% RSLogix 500 project Backwash Alarm Control and Interlock System.RSS, saved by version 9.00.00.04 %
PROJECT "SAMPLE2"    % processor: MicroLogix 1400 %

PROGRAM FILES
  LAD 2 "MAIN"  21 rungs
  LAD 3 "REGEN"  29 rungs
  LAD 4 "FLOW AB"  43 rungs
  LAD 5 "ALARMS"  22 rungs
  LAD 6 "TIME TRIG"  17 rungs  % TIME INTERVAL REGN INITIATION %
  LAD 7 "A VESSEL"  38 rungs
  LAD 8 "ANALOG IN"  6 rungs
  LAD 9 "PRESSURE"  11 rungs
  LAD 10 "B VESSEL"  38 rungs
  LAD 11 "DIGITAL IN"  4 rungs
  LAD 12 "WELL PUMP"  4 rungs
  LAD 16 "DIGITL OUT"  15 rungs
  LAD 17 "REGEN A"  17 rungs
  LAD 18 "REGEN B"  17 rungs
  LAD 19 "RECYCLE"  17 rungs

DATA FILES
  O0 OUTPUT  7 elements
  I1 INPUT  22 elements
  S2 STATUS  66 elements
  B3 COMMON  14 elements
  T4 TIMER  56 elements
  C5 COUNTER  13 elements
  R6 CONTROL  1 elements
  N7   52 elements
  F8 FLOAT  122 elements
  B9 GENCTRL  3 elements
  C10   5 elements
  B21 A  BITS  7 elements
  B22 B BITS  7 elements
  N34   92 elements

LADDER 2 "MAIN"
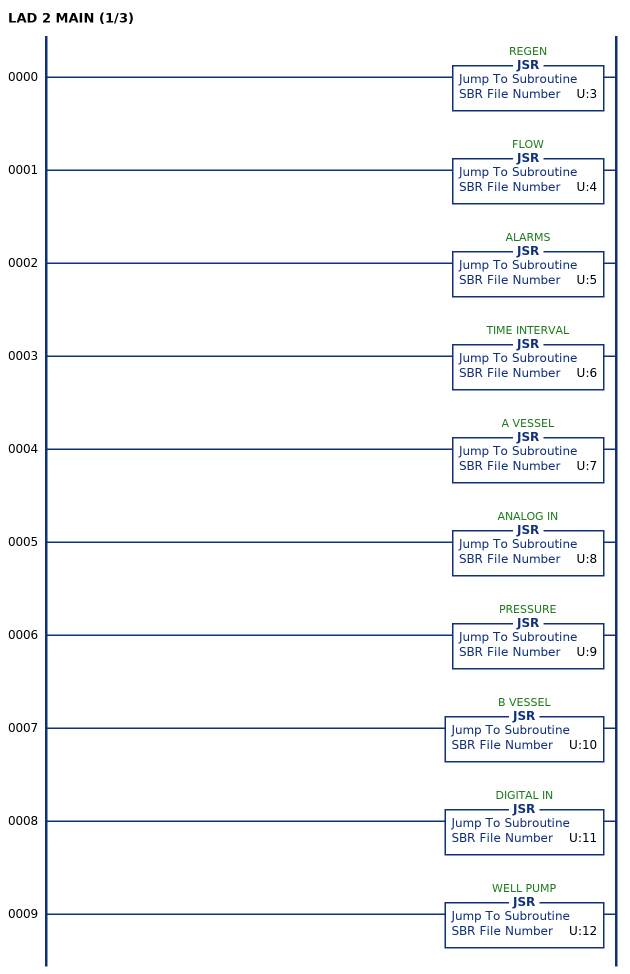
% Rung: 0 %
SOR JSR U:3 EOR
%   U:3  "REGEN" %
% Rung: 1 %
SOR JSR U:4 EOR
%   U:4  "FLOW" %
% Rung: 2 %
SOR JSR U:5 EOR
%   U:5  "ALARMS" %
% Rung: 3 %
SOR JSR U:6 EOR
%   U:6  "TIME INTERVAL" %
% Rung: 4 %
SOR JSR U:7 EOR
%   U:7  "A VESSEL" %
% Rung: 5 %
SOR JSR U:8 EOR
%   U:8  "ANALOG IN" %
% Rung: 6 %
SOR JSR U:9 EOR
%   U:9  "PRESSURE" %
% Rung: 7 %
SOR JSR U:10 EOR
%   U:10  "B VESSEL" %
% Rung: 8 %
SOR JSR U:11 EOR
%   U:11  "DIGITAL IN" %
% Rung: 9 %
SOR JSR U:12 EOR
%   U:12  "WELL PUMP" %

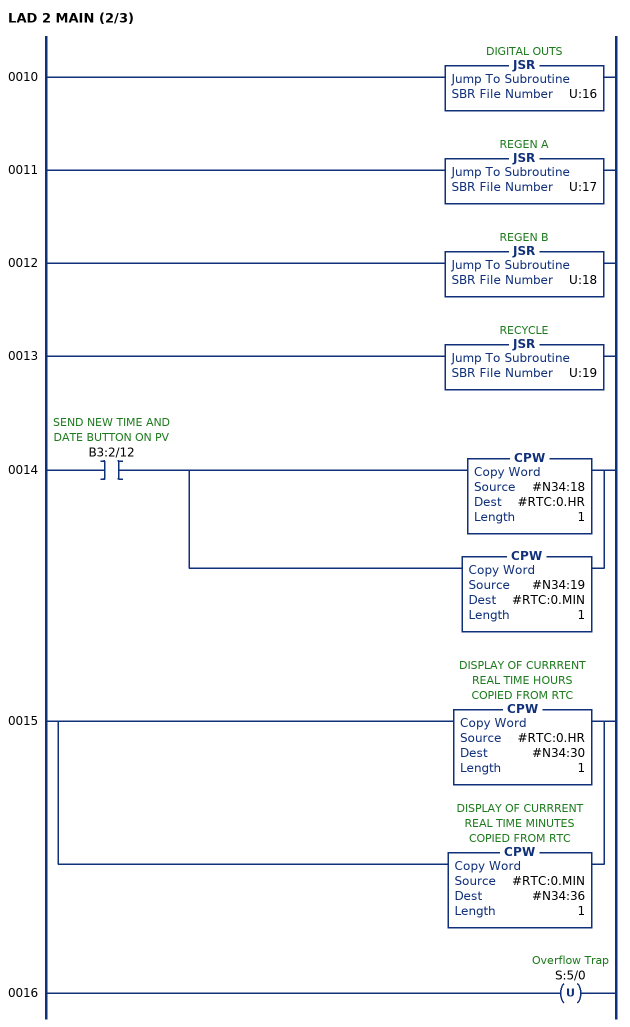
% Rung: 10 %
SOR JSR U:16 EOR
%   U:16  "DIGITAL OUTS" %
% Rung: 11 %
SOR JSR U:17 EOR
%   U:17  "REGEN A" %
% Rung: 12 %
SOR JSR U:18 EOR
%   U:18  "REGEN B" %
% Rung: 13 %
SOR JSR U:19 EOR
%   U:19  "RECYCLE" %
% Rung: 14 %
SOR XIC B3:2/12 BST CPW #N34:18 #RTC:0.HR 1 NXB CPW #N34:19 #RTC:0.MIN 1 BND EOR
%   B3:2/12  "SEND NEW TIME AND DATE BUTTON ON PV" %
%   N34:18  "HOUR INPUT FROM PV" %
%   N34:19  "MINUTE INPUT FROM PV" %
% Rung: 15 %
SOR BST CPW #RTC:0.HR #N34:30 1 NXB CPW #RTC:0.MIN #N34:36 1 BND EOR
%   N34:30  "DISPLAY OF CURRRENT REAL TIME HOURS COPIED FROM RTC" %
%   N34:36  "DISPLAY OF CURRRENT REAL TIME MINUTES COPIED FROM RTC" %
% Rung: 16 %
SOR OTU S:5/0 EOR
%   S:5/0  "Overflow Trap" %

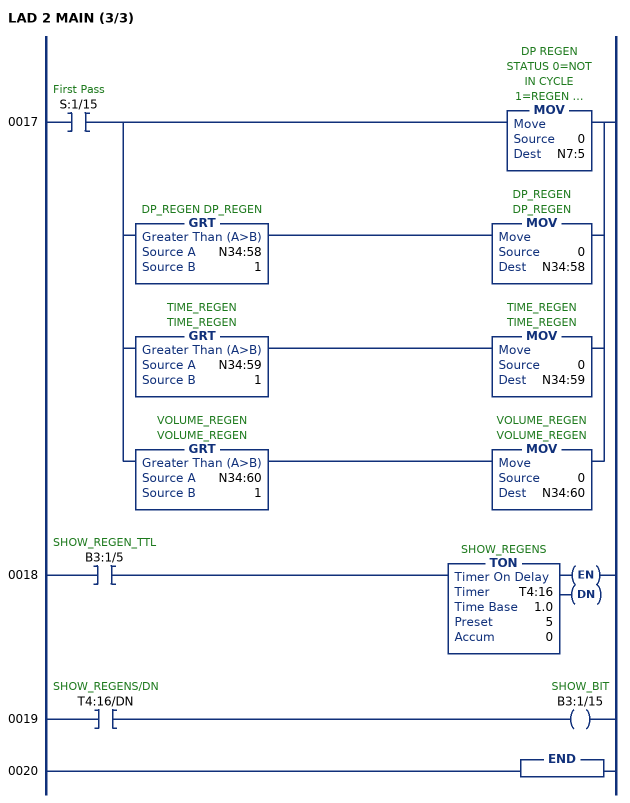
% Rung: 17 %
SOR XIC S:1/15 BST MOV 0 N7:5 NXB GRT N34:58 1 MOV 0 N34:58 NXB GRT N34:59 1 MOV 0 N34:59 NXB GRT N34:60 1 MOV 0 N34:60 BND EOR
%   S:1/15  "First Pass" %
%   N7:5  "DP REGEN STATUS 0=NOT IN CYCLE 1=REGEN A 2=REGEN B" %
%   N34:58  DP_REGEN  "DP_REGEN" %
%   N34:59  TIME_REGEN  "TIME_REGEN" %
%   N34:60  VOLUME_REGEN  "VOLUME_REGEN" %
% Rung: 18 %
SOR XIC B3:1/5 TON T4:16 1.0 5 0 EOR
%   B3:1/5  SHOW_REGEN_TTL %
%   T4:16  SHOW_REGENS %
% Rung: 19 %
SOR XIC T4:16/DN OTE B3:1/15 EOR
%   T4:16  SHOW_REGENS %
%   B3:1/15  SHOW_BIT %
% Rung: 20 %
SOR END EOR

LADDER 3 "REGEN"
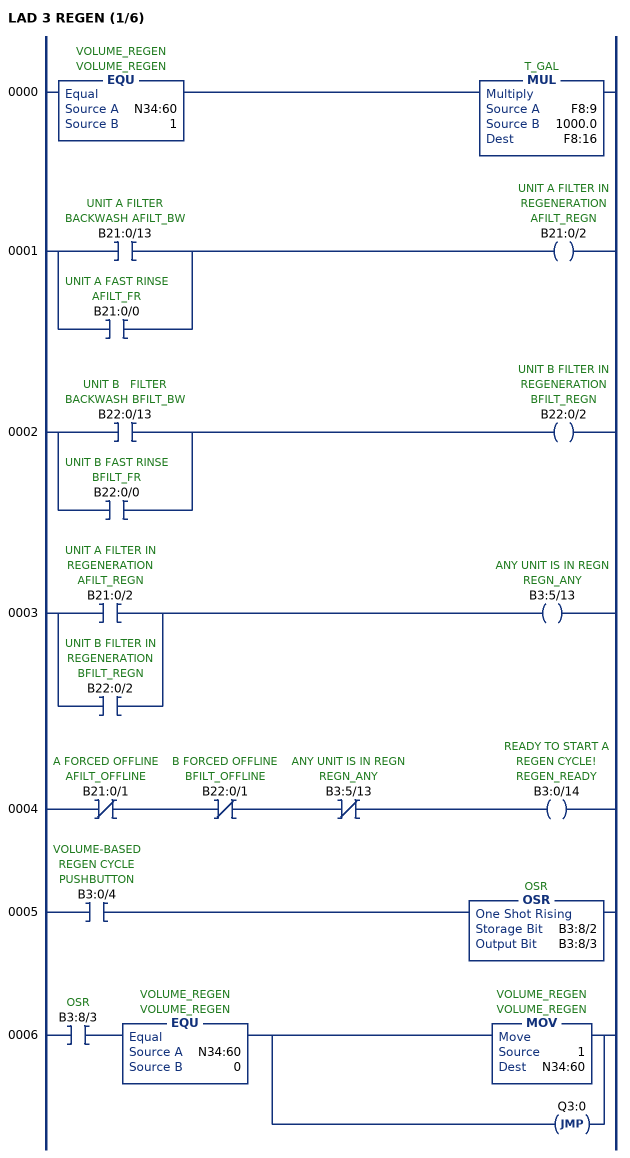
% Rung: 0 %
SOR EQU N34:60 1 MUL F8:9 1000.0 F8:16 EOR
%   N34:60  VOLUME_REGEN  "VOLUME_REGEN" %
%   F8:9  "BATCH ENTRY FOR BATCH START" %
%   F8:16  T_GAL %
% Rung: 1 %
SOR BST XIC B21:0/13 NXB XIC B21:0/0 BND OTE B21:0/2 EOR
%   B21:0/13  AFILT_BW  "UNIT A FILTER BACKWASH" %
%   B21:0/0  AFILT_FR  "UNIT A FAST RINSE" %
%   B21:0/2  AFILT_REGN  "UNIT A FILTER IN REGENERATION" %
% Rung: 2 %
SOR BST XIC B22:0/13 NXB XIC B22:0/0 BND OTE B22:0/2 EOR
%   B22:0/13  BFILT_BW  "UNIT B   FILTER BACKWASH" %
%   B22:0/0  BFILT_FR  "UNIT B FAST RINSE" %
%   B22:0/2  BFILT_REGN  "UNIT B FILTER IN REGENERATION" %
% Rung: 3 %
SOR BST XIC B21:0/2 NXB XIC B22:0/2 BND OTE B3:5/13 EOR
%   B21:0/2  AFILT_REGN  "UNIT A FILTER IN REGENERATION" %
%   B22:0/2  BFILT_REGN  "UNIT B FILTER IN REGENERATION" %
%   B3:5/13  REGN_ANY  "ANY UNIT IS IN REGN" %
% Rung: 4 %
SOR XIO B21:0/1 XIO B22:0/1 XIO B3:5/13 OTE B3:0/14 EOR
%   B21:0/1  AFILT_OFFLINE  "A FORCED OFFLINE" %
%   B22:0/1  BFILT_OFFLINE  "B FORCED OFFLINE" %
%   B3:5/13  REGN_ANY  "ANY UNIT IS IN REGN" %
%   B3:0/14  REGEN_READY  "READY TO START A REGEN CYCLE!" %
% Rung: 5 %
SOR XIC B3:0/4 OSR B3:8/2 B3:8/3 EOR
%   B3:0/4  "VOLUME-BASED REGEN CYCLE PUSHBUTTON" %
%   B3:8/2  "OSR" %
%   B3:8/3  "OSR" %
% Rung: 6 %
SOR XIC B3:8/3 EQU N34:60 0 BST MOV 1 N34:60 NXB JMP Q3:0 BND EOR
%   B3:8/3  "OSR" %
%   N34:60  VOLUME_REGEN  "VOLUME_REGEN" %

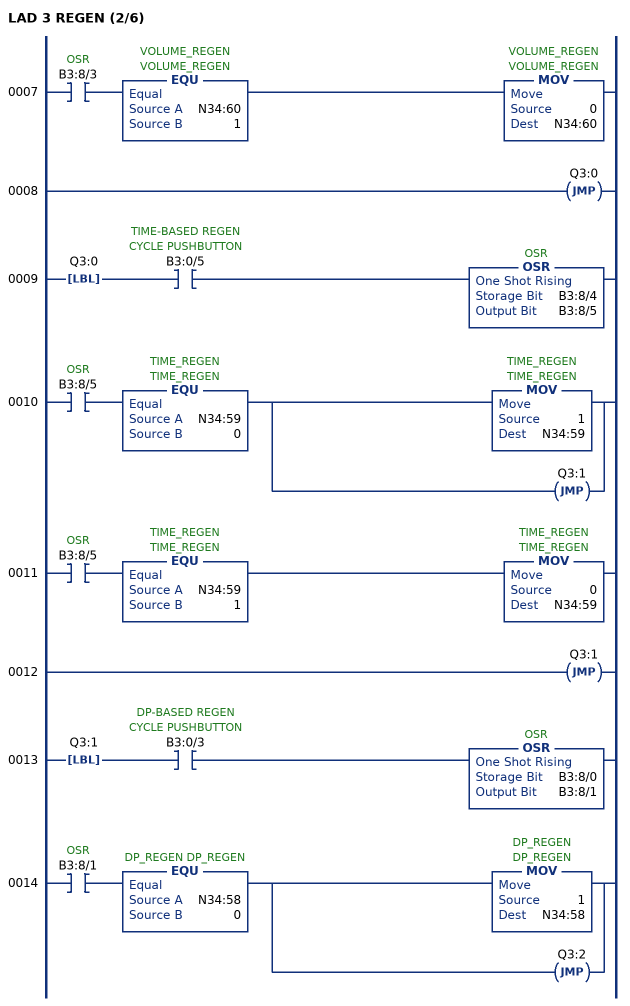
% Rung: 7 %
SOR XIC B3:8/3 EQU N34:60 1 MOV 0 N34:60 EOR
%   B3:8/3  "OSR" %
%   N34:60  VOLUME_REGEN  "VOLUME_REGEN" %
% Rung: 8 %
SOR JMP Q3:0 EOR
% Rung: 9 %
SOR LBL Q3:0 XIC B3:0/5 OSR B3:8/4 B3:8/5 EOR
%   B3:0/5  "TIME-BASED REGEN CYCLE PUSHBUTTON" %
%   B3:8/4  "OSR" %
%   B3:8/5  "OSR" %
% Rung: 10 %
SOR XIC B3:8/5 EQU N34:59 0 BST MOV 1 N34:59 NXB JMP Q3:1 BND EOR
%   B3:8/5  "OSR" %
%   N34:59  TIME_REGEN  "TIME_REGEN" %
% Rung: 11 %
SOR XIC B3:8/5 EQU N34:59 1 MOV 0 N34:59 EOR
%   B3:8/5  "OSR" %
%   N34:59  TIME_REGEN  "TIME_REGEN" %
% Rung: 12 %
SOR JMP Q3:1 EOR
% Rung: 13 %
SOR LBL Q3:1 XIC B3:0/3 OSR B3:8/0 B3:8/1 EOR
%   B3:0/3  "DP-BASED REGEN CYCLE PUSHBUTTON" %
%   B3:8/0  "OSR" %
%   B3:8/1  "OSR" %
% Rung: 14 %
SOR XIC B3:8/1 EQU N34:58 0 BST MOV 1 N34:58 NXB JMP Q3:2 BND EOR
%   B3:8/1  "OSR" %
%   N34:58  DP_REGEN  "DP_REGEN" %

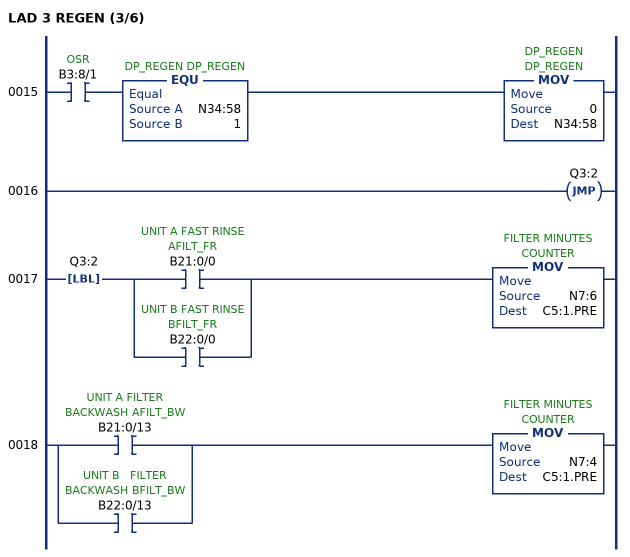
% Rung: 15 %
SOR XIC B3:8/1 EQU N34:58 1 MOV 0 N34:58 EOR
%   B3:8/1  "OSR" %
%   N34:58  DP_REGEN  "DP_REGEN" %
% Rung: 16 %
SOR JMP Q3:2 EOR
% Rung: 17 %
SOR LBL Q3:2 BST XIC B21:0/0 NXB XIC B22:0/0 BND MOV N7:6 C5:1.PRE EOR
%   B21:0/0  AFILT_FR  "UNIT A FAST RINSE" %
%   B22:0/0  BFILT_FR  "UNIT B FAST RINSE" %
%   N7:6  "FILTER FAST RINSE ENTRY FROM OIT" %
%   C5:1.PRE  "FILTER MINUTES COUNTER" %
% Rung: 18 %
SOR BST XIC B21:0/13 NXB XIC B22:0/13 BND MOV N7:4 C5:1.PRE EOR
%   B21:0/13  AFILT_BW  "UNIT A FILTER BACKWASH" %
%   B22:0/13  BFILT_BW  "UNIT B   FILTER BACKWASH" %
%   N7:4  "FILTER BACKWASH PRE FROM OIT" %
%   C5:1.PRE  "FILTER MINUTES COUNTER" %

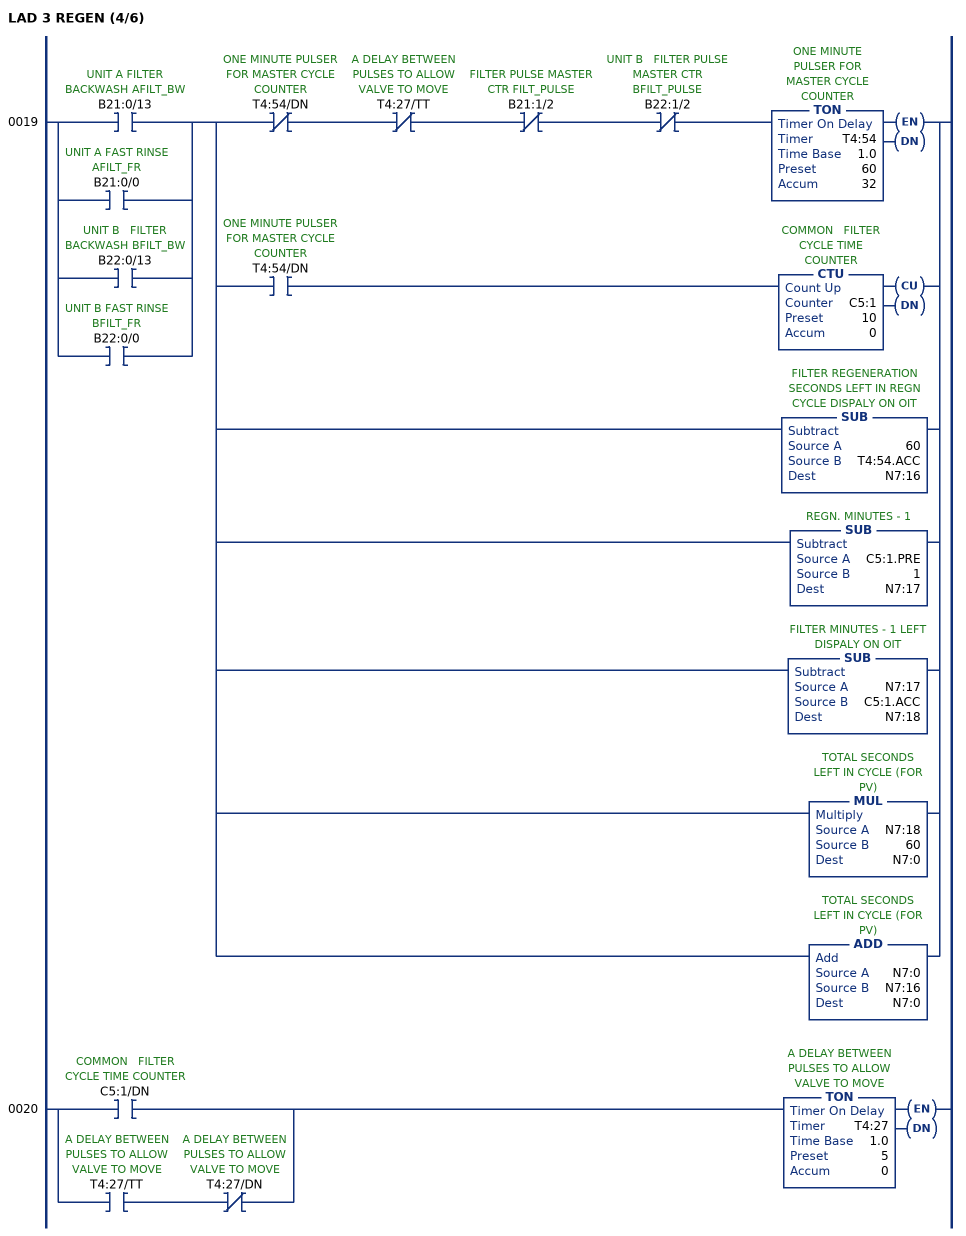
% Rung: 19 %
SOR BST XIC B21:0/13 NXB XIC B21:0/0 NXB XIC B22:0/13 NXB XIC B22:0/0 BND BST XIO T4:54/DN XIO T4:27/TT XIO B21:1/2 XIO B22:1/2 TON T4:54 1.0 60 32 NXB XIC T4:54/DN CTU C5:1 10 0 NXB SUB 60 T4:54.ACC N7:16 NXB SUB C5:1.PRE 1 N7:17 NXB SUB N7:17 C5:1.ACC N7:18 NXB MUL N7:18 60 N7:0 NXB ADD N7:0 N7:16 N7:0 BND EOR
%   B21:0/13  AFILT_BW  "UNIT A FILTER BACKWASH" %
%   B21:0/0  AFILT_FR  "UNIT A FAST RINSE" %
%   B22:0/13  BFILT_BW  "UNIT B   FILTER BACKWASH" %
%   B22:0/0  BFILT_FR  "UNIT B FAST RINSE" %
%   T4:54  "ONE MINUTE PULSER FOR MASTER CYCLE COUNTER" %
%   T4:27  "A DELAY BETWEEN PULSES TO ALLOW VALVE TO MOVE" %
%   B21:1/2  FILT_PULSE  "FILTER PULSE MASTER CTR" %
%   B22:1/2  BFILT_PULSE  "UNIT B   FILTER PULSE MASTER CTR" %
%   C5:1  "COMMON   FILTER CYCLE TIME COUNTER" %
%   N7:16  "FILTER REGENERATION SECONDS LEFT IN REGN CYCLE DISPALY ON OIT" %
%   C5:1.PRE  "FILTER MINUTES COUNTER" %
%   N7:17  "REGN. MINUTES - 1" %
%   N7:18  "FILTER MINUTES - 1 LEFT DISPALY ON OIT" %
%   N7:0  "TOTAL SECONDS LEFT IN CYCLE (FOR PV)" %
% Rung: 20 %
SOR BST XIC C5:1/DN NXB XIC T4:27/TT XIO T4:27/DN BND TON T4:27 1.0 5 0 EOR
%   C5:1  "COMMON   FILTER CYCLE TIME COUNTER" %
%   T4:27  "A DELAY BETWEEN PULSES TO ALLOW VALVE TO MOVE" %

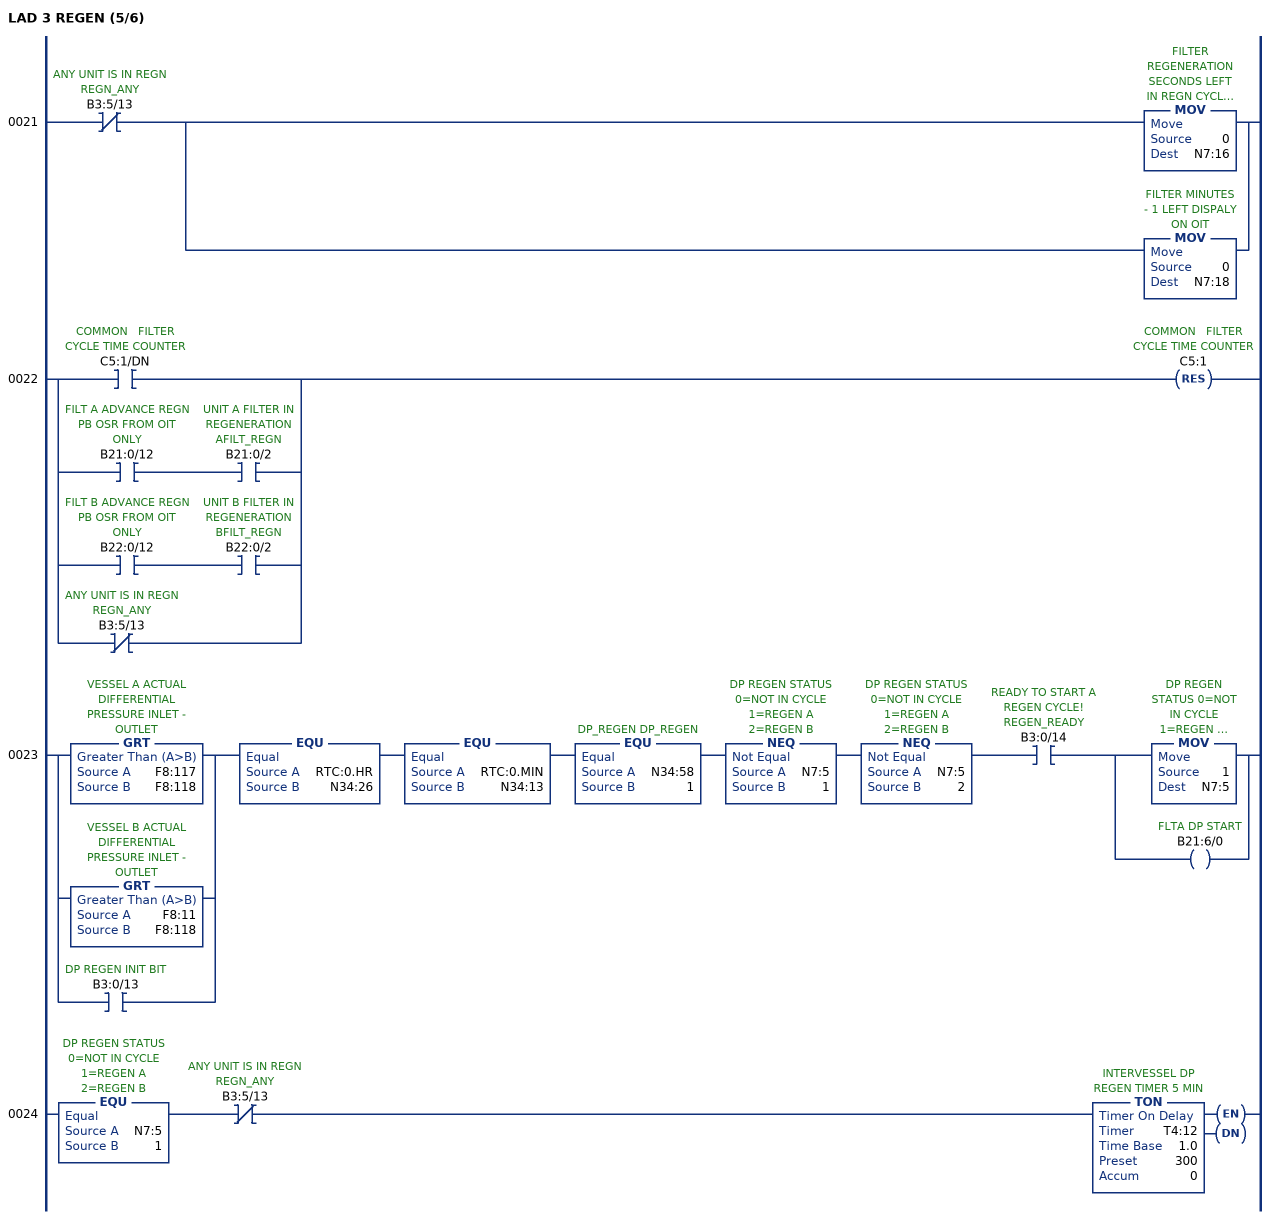
% Rung: 21 %
SOR XIO B3:5/13 BST MOV 0 N7:16 NXB MOV 0 N7:18 BND EOR
%   B3:5/13  REGN_ANY  "ANY UNIT IS IN REGN" %
%   N7:16  "FILTER REGENERATION SECONDS LEFT IN REGN CYCLE DISPALY ON OIT" %
%   N7:18  "FILTER MINUTES - 1 LEFT DISPALY ON OIT" %
% Rung: 22 %
SOR BST XIC C5:1/DN NXB XIC B21:0/12 XIC B21:0/2 NXB XIC B22:0/12 XIC B22:0/2 NXB XIO B3:5/13 BND RES C5:1 EOR
%   C5:1  "COMMON   FILTER CYCLE TIME COUNTER" %
%   B21:0/12  "FILT A ADVANCE REGN PB OSR FROM OIT ONLY" %
%   B21:0/2  AFILT_REGN  "UNIT A FILTER IN REGENERATION" %
%   B22:0/12  "FILT B ADVANCE REGN PB OSR FROM OIT ONLY" %
%   B22:0/2  BFILT_REGN  "UNIT B FILTER IN REGENERATION" %
%   B3:5/13  REGN_ANY  "ANY UNIT IS IN REGN" %
% Rung: 23 %
SOR BST BST GRT F8:117 F8:118 NXB GRT F8:11 F8:118 BND NXB XIC B3:0/13 BND EQU RTC:0.HR N34:26 EQU RTC:0.MIN N34:13 EQU N34:58 1 NEQ N7:5 1 NEQ N7:5 2 XIC B3:0/14 BST MOV 1 N7:5 NXB OTE B21:6/0 BND EOR
%   F8:117  "VESSEL A ACTUAL DIFFERENTIAL PRESSURE INLET - OUTLET" %
%   F8:118  DP_SETPOINT  "PRESSURE DIFFERENTIAL SETPOINT" %
%   F8:11  "VESSEL B ACTUAL DIFFERENTIAL PRESSURE INLET - OUTLET" %
%   B3:0/13  "DP REGEN INIT BIT" %
%   N34:26  "FILTER A HOUR OF DAY TO START SELECT EITHER DUE TO BATCH OR ELAPSED TIME OR DP" %
%   N34:13  "FILTER A MIN OF DAY TO START SELECT EITHER DUE TO BATCH OR ELAPSED TIME" %
%   N34:58  DP_REGEN  "DP_REGEN" %
%   N7:5  "DP REGEN STATUS 0=NOT IN CYCLE 1=REGEN A 2=REGEN B" %
%   B3:0/14  REGEN_READY  "READY TO START A REGEN CYCLE!" %
%   B21:6/0  "FLTA DP START" %
% Rung: 24 %
SOR EQU N7:5 1 XIO B3:5/13 TON T4:12 1.0 300 0 EOR
%   N7:5  "DP REGEN STATUS 0=NOT IN CYCLE 1=REGEN A 2=REGEN B" %
%   B3:5/13  REGN_ANY  "ANY UNIT IS IN REGN" %
%   T4:12  "INTERVESSEL DP REGEN TIMER 5 MIN" %

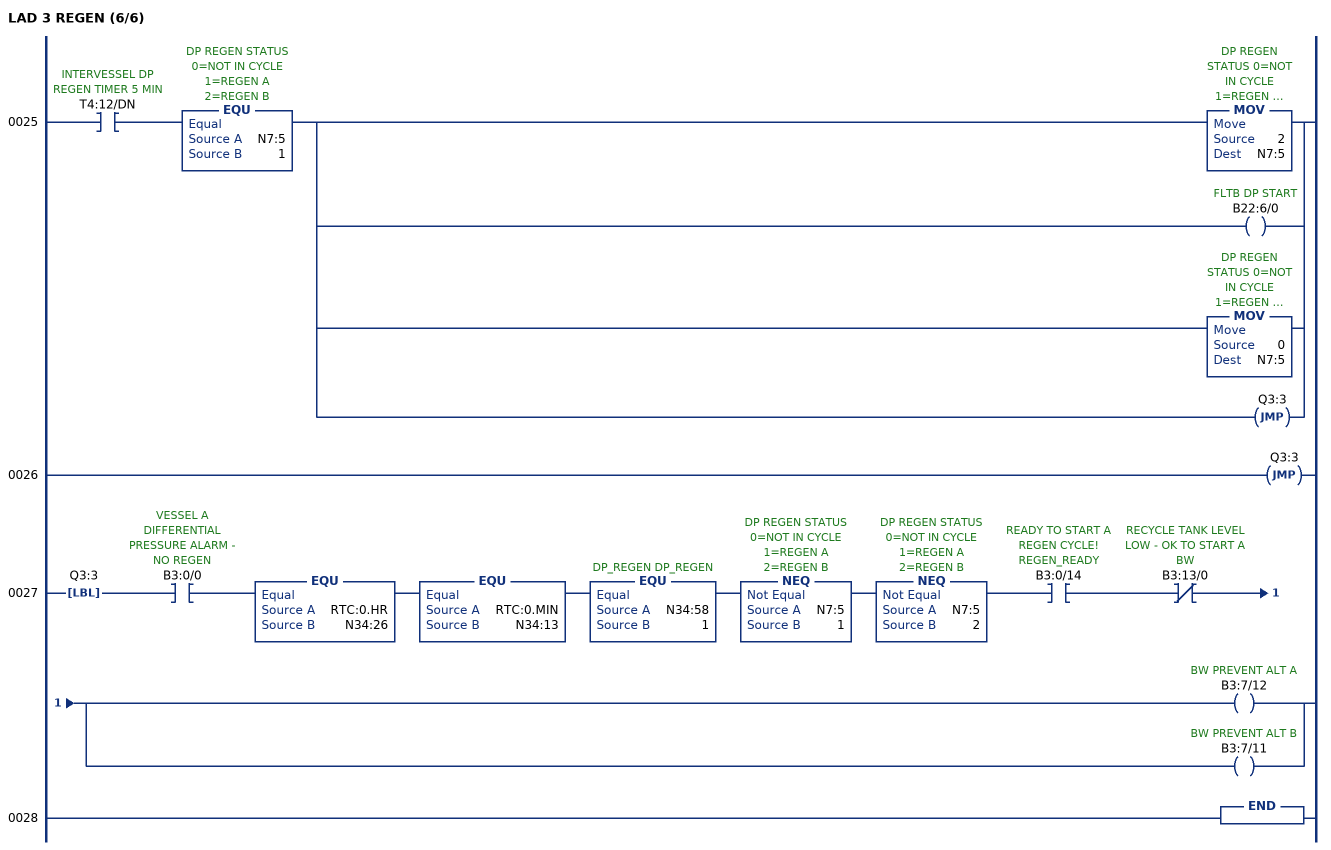
% Rung: 25 %
SOR XIC T4:12/DN EQU N7:5 1 BST MOV 2 N7:5 NXB OTE B22:6/0 NXB MOV 0 N7:5 NXB JMP Q3:3 BND EOR
%   T4:12  "INTERVESSEL DP REGEN TIMER 5 MIN" %
%   N7:5  "DP REGEN STATUS 0=NOT IN CYCLE 1=REGEN A 2=REGEN B" %
%   B22:6/0  "FLTB DP START" %
% Rung: 26 %
SOR JMP Q3:3 EOR
% Rung: 27 %
SOR LBL Q3:3 XIC B3:0/0 EQU RTC:0.HR N34:26 EQU RTC:0.MIN N34:13 EQU N34:58 1 NEQ N7:5 1 NEQ N7:5 2 XIC B3:0/14 XIO B3:13/0 BST OTE B3:7/12 NXB OTE B3:7/11 BND EOR
%   B3:0/0  "VESSEL A DIFFERENTIAL PRESSURE ALARM - NO REGEN" %
%   N34:26  "FILTER A HOUR OF DAY TO START SELECT EITHER DUE TO BATCH OR ELAPSED TIME OR DP" %
%   N34:13  "FILTER A MIN OF DAY TO START SELECT EITHER DUE TO BATCH OR ELAPSED TIME" %
%   N34:58  DP_REGEN  "DP_REGEN" %
%   N7:5  "DP REGEN STATUS 0=NOT IN CYCLE 1=REGEN A 2=REGEN B" %
%   B3:0/14  REGEN_READY  "READY TO START A REGEN CYCLE!" %
%   B3:13/0  "RECYCLE TANK LEVEL LOW - OK TO START A BW" %
%   B3:7/12  "BW PREVENT ALT A" %
%   B3:7/11  "BW PREVENT ALT B" %
% Rung: 28 %
SOR END EOR

LADDER 4 "FLOW AB"
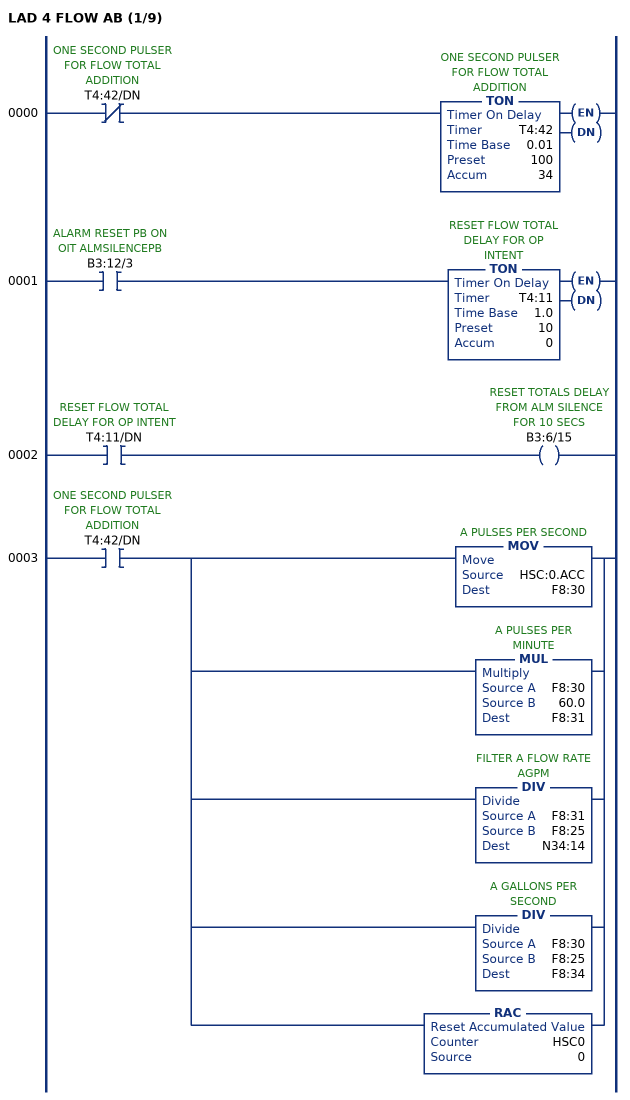
% Rung: 0 %
SOR XIO T4:42/DN TON T4:42 0.01 100 34 EOR
%   T4:42  "ONE SECOND PULSER FOR FLOW TOTAL ADDITION" %
% Rung: 1 %
SOR XIC B3:12/3 TON T4:11 1.0 10 0 EOR
%   B3:12/3  ALMSILENCEPB  "ALARM RESET PB ON OIT" %
%   T4:11  "RESET FLOW TOTAL DELAY FOR OP INTENT" %
% Rung: 2 %
SOR XIC T4:11/DN OTE B3:6/15 EOR
%   T4:11  "RESET FLOW TOTAL DELAY FOR OP INTENT" %
%   B3:6/15  "RESET TOTALS DELAY FROM ALM SILENCE FOR 10 SECS" %
% Rung: 3 %
SOR XIC T4:42/DN BST MOV HSC:0.ACC F8:30 NXB MUL F8:30 60.0 F8:31 NXB DIV F8:31 F8:25 N34:14 NXB DIV F8:30 F8:25 F8:34 NXB RAC HSC0 0 BND EOR
%   T4:42  "ONE SECOND PULSER FOR FLOW TOTAL ADDITION" %
%   F8:30  "A PULSES PER SECOND" %
%   F8:31  "A PULSES PER MINUTE" %
%   F8:25  "CHEM1 GALLONS PER PULSE" %
%   N34:14  AGPM  "FILTER A FLOW RATE" %
%   F8:34  "A GALLONS PER SECOND" %

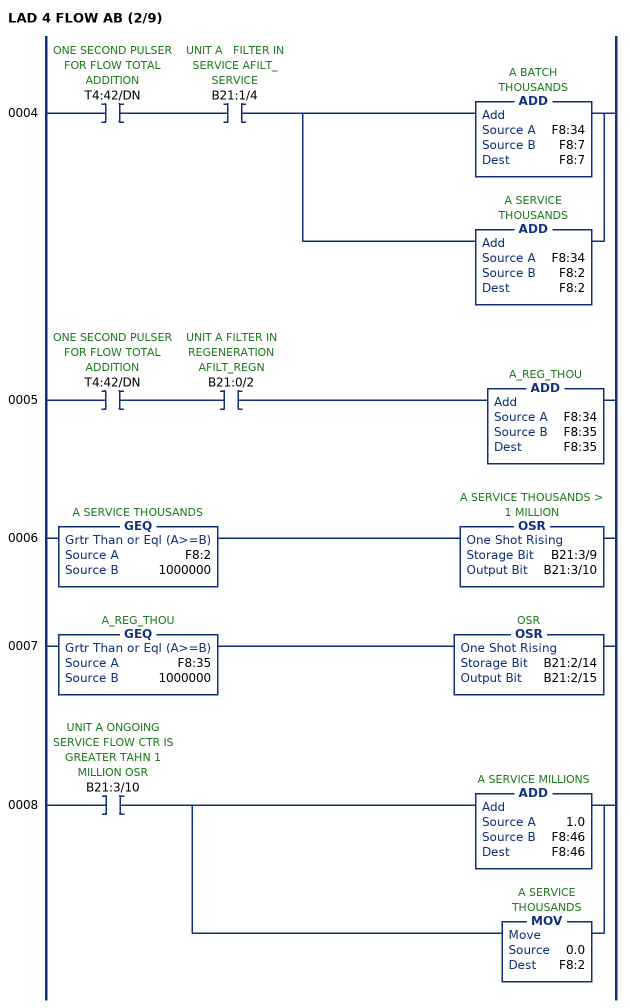
% Rung: 4 %
SOR XIC T4:42/DN XIC B21:1/4 BST ADD F8:34 F8:7 F8:7 NXB ADD F8:34 F8:2 F8:2 BND EOR
%   T4:42  "ONE SECOND PULSER FOR FLOW TOTAL ADDITION" %
%   B21:1/4  AFILT_SERVICE  "UNIT A   FILTER IN SERVICE" %
%   F8:34  "A GALLONS PER SECOND" %
%   F8:7  "A BATCH THOUSANDS" %
%   F8:2  "A SERVICE THOUSANDS" %
% Rung: 5 %
SOR XIC T4:42/DN XIC B21:0/2 ADD F8:34 F8:35 F8:35 EOR
%   T4:42  "ONE SECOND PULSER FOR FLOW TOTAL ADDITION" %
%   B21:0/2  AFILT_REGN  "UNIT A FILTER IN REGENERATION" %
%   F8:34  "A GALLONS PER SECOND" %
%   F8:35  A_REG_THOU %
% Rung: 6 %
SOR GEQ F8:2 1000000 OSR B21:3/9 B21:3/10 EOR
%   F8:2  "A SERVICE THOUSANDS" %
%   B21:3/9  "A SERVICE THOUSANDS > 1 MILLION" %
%   B21:3/10  "UNIT A ONGOING SERVICE FLOW CTR IS GREATER TAHN 1 MILLION OSR" %
% Rung: 7 %
SOR GEQ F8:35 1000000 OSR B21:2/14 B21:2/15 EOR
%   F8:35  A_REG_THOU %
%   B21:2/14  "OSR" %
%   B21:2/15  "OSR" %
% Rung: 8 %
SOR XIC B21:3/10 BST ADD 1.0 F8:46 F8:46 NXB MOV 0.0 F8:2 BND EOR
%   B21:3/10  "UNIT A ONGOING SERVICE FLOW CTR IS GREATER TAHN 1 MILLION OSR" %
%   F8:46  "A SERVICE MILLIONS" %
%   F8:2  "A SERVICE THOUSANDS" %

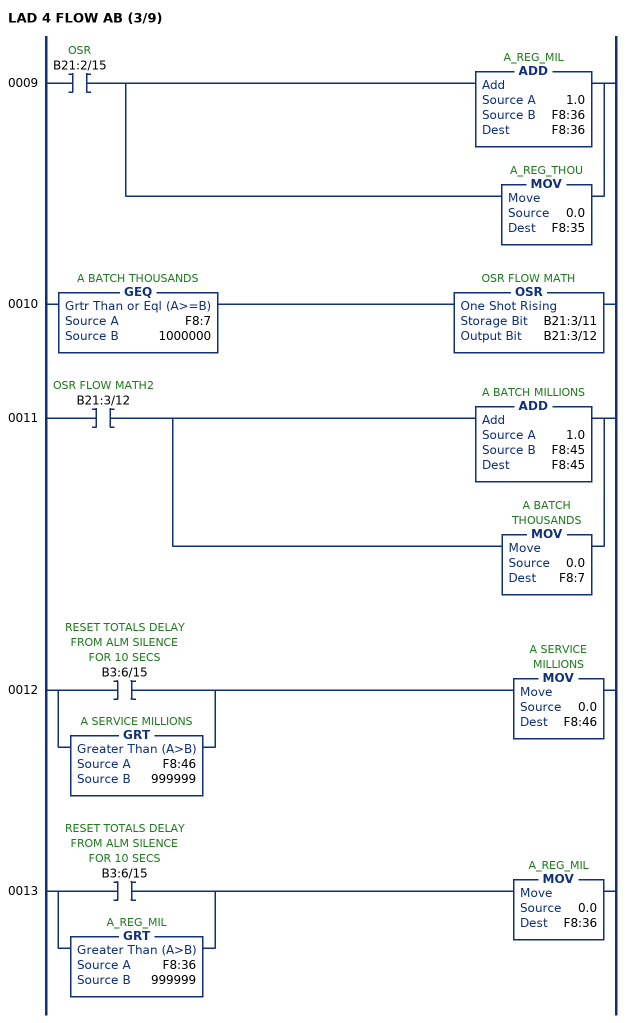
% Rung: 9 %
SOR XIC B21:2/15 BST ADD 1.0 F8:36 F8:36 NXB MOV 0.0 F8:35 BND EOR
%   B21:2/15  "OSR" %
%   F8:36  A_REG_MIL %
%   F8:35  A_REG_THOU %
% Rung: 10 %
SOR GEQ F8:7 1000000 OSR B21:3/11 B21:3/12 EOR
%   F8:7  "A BATCH THOUSANDS" %
%   B21:3/11  "OSR FLOW MATH" %
%   B21:3/12  "OSR FLOW MATH2" %
% Rung: 11 %
SOR XIC B21:3/12 BST ADD 1.0 F8:45 F8:45 NXB MOV 0.0 F8:7 BND EOR
%   B21:3/12  "OSR FLOW MATH2" %
%   F8:45  "A BATCH MILLIONS" %
%   F8:7  "A BATCH THOUSANDS" %
% Rung: 12 %
SOR BST XIC B3:6/15 NXB GRT F8:46 999999 BND MOV 0.0 F8:46 EOR
%   B3:6/15  "RESET TOTALS DELAY FROM ALM SILENCE FOR 10 SECS" %
%   F8:46  "A SERVICE MILLIONS" %
% Rung: 13 %
SOR BST XIC B3:6/15 NXB GRT F8:36 999999 BND MOV 0.0 F8:36 EOR
%   B3:6/15  "RESET TOTALS DELAY FROM ALM SILENCE FOR 10 SECS" %
%   F8:36  A_REG_MIL %

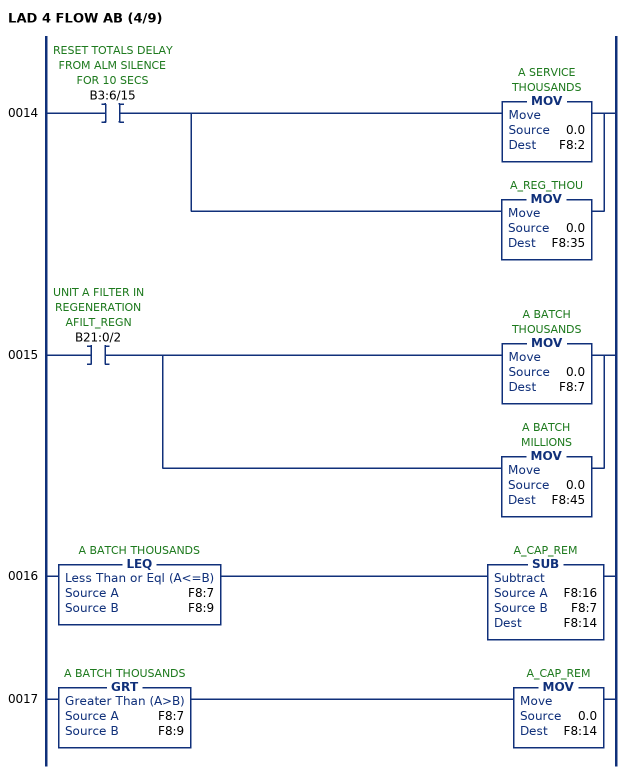
% Rung: 14 %
SOR XIC B3:6/15 BST MOV 0.0 F8:2 NXB MOV 0.0 F8:35 BND EOR
%   B3:6/15  "RESET TOTALS DELAY FROM ALM SILENCE FOR 10 SECS" %
%   F8:2  "A SERVICE THOUSANDS" %
%   F8:35  A_REG_THOU %
% Rung: 15 %
SOR XIC B21:0/2 BST MOV 0.0 F8:7 NXB MOV 0.0 F8:45 BND EOR
%   B21:0/2  AFILT_REGN  "UNIT A FILTER IN REGENERATION" %
%   F8:7  "A BATCH THOUSANDS" %
%   F8:45  "A BATCH MILLIONS" %
% Rung: 16 %
SOR LEQ F8:7 F8:9 SUB F8:16 F8:7 F8:14 EOR
%   F8:7  "A BATCH THOUSANDS" %
%   F8:9  "BATCH ENTRY FOR BATCH START" %
%   F8:16  T_GAL %
%   F8:14  A_CAP_REM %
% Rung: 17 %
SOR GRT F8:7 F8:9 MOV 0.0 F8:14 EOR
%   F8:7  "A BATCH THOUSANDS" %
%   F8:9  "BATCH ENTRY FOR BATCH START" %
%   F8:14  A_CAP_REM %

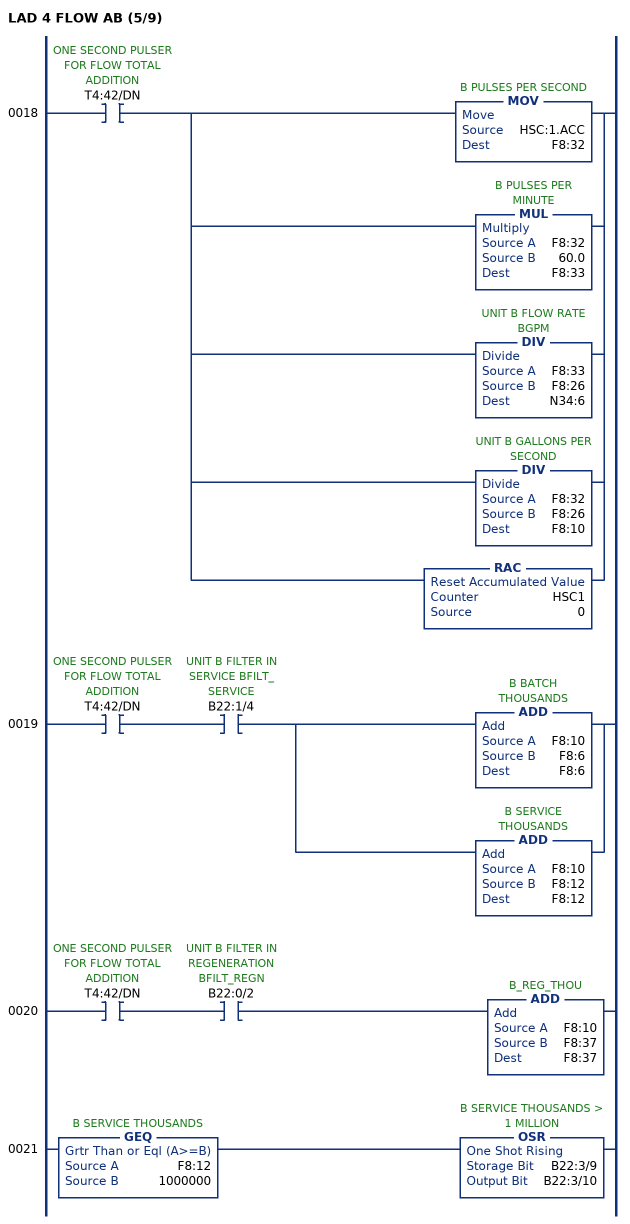
% Rung: 18 %
SOR XIC T4:42/DN BST MOV HSC:1.ACC F8:32 NXB MUL F8:32 60.0 F8:33 NXB DIV F8:33 F8:26 N34:6 NXB DIV F8:32 F8:26 F8:10 NXB RAC HSC1 0 BND EOR
%   T4:42  "ONE SECOND PULSER FOR FLOW TOTAL ADDITION" %
%   F8:32  "B PULSES PER SECOND" %
%   F8:33  "B PULSES PER MINUTE" %
%   F8:26  "B K FACTOR" %
%   N34:6  BGPM  "UNIT B FLOW RATE" %
%   F8:10  "UNIT B GALLONS PER SECOND" %
% Rung: 19 %
SOR XIC T4:42/DN XIC B22:1/4 BST ADD F8:10 F8:6 F8:6 NXB ADD F8:10 F8:12 F8:12 BND EOR
%   T4:42  "ONE SECOND PULSER FOR FLOW TOTAL ADDITION" %
%   B22:1/4  BFILT_SERVICE  "UNIT B FILTER IN SERVICE" %
%   F8:10  "UNIT B GALLONS PER SECOND" %
%   F8:6  "B BATCH THOUSANDS" %
%   F8:12  "B SERVICE THOUSANDS" %
% Rung: 20 %
SOR XIC T4:42/DN XIC B22:0/2 ADD F8:10 F8:37 F8:37 EOR
%   T4:42  "ONE SECOND PULSER FOR FLOW TOTAL ADDITION" %
%   B22:0/2  BFILT_REGN  "UNIT B FILTER IN REGENERATION" %
%   F8:10  "UNIT B GALLONS PER SECOND" %
%   F8:37  B_REG_THOU %
% Rung: 21 %
SOR GEQ F8:12 1000000 OSR B22:3/9 B22:3/10 EOR
%   F8:12  "B SERVICE THOUSANDS" %
%   B22:3/9  "B SERVICE THOUSANDS > 1 MILLION" %
%   B22:3/10  "UNIT B ONGOING SERVICE FLOW CTR IS GREATER THAN 1 MILLION OSR" %

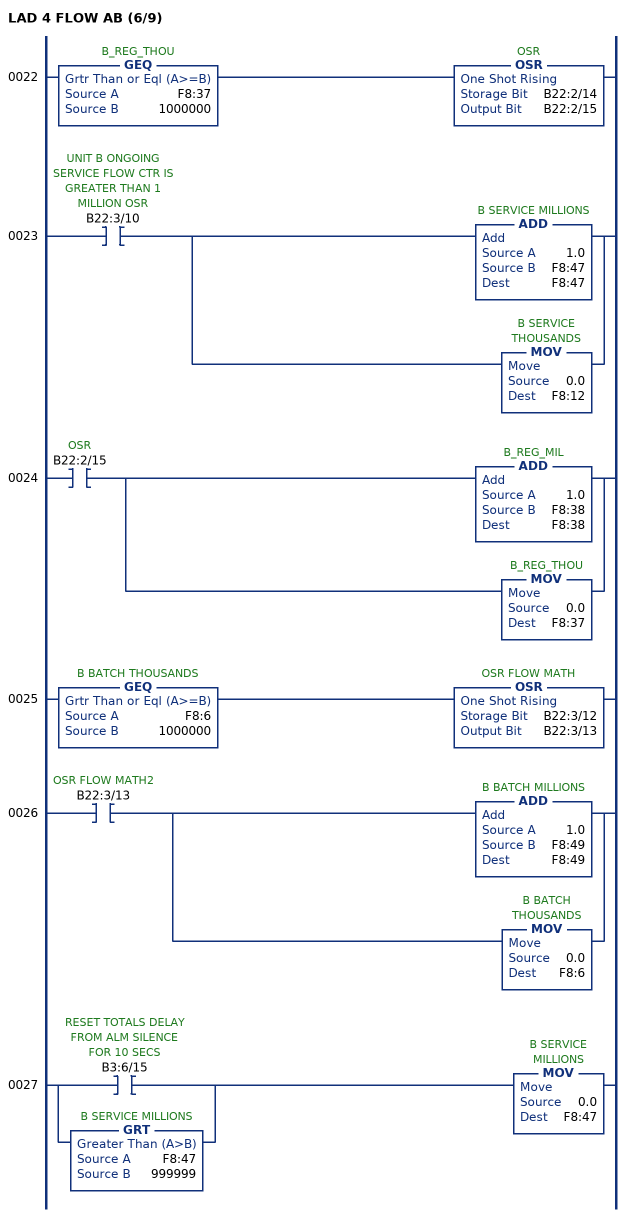
% Rung: 22 %
SOR GEQ F8:37 1000000 OSR B22:2/14 B22:2/15 EOR
%   F8:37  B_REG_THOU %
%   B22:2/14  "OSR" %
%   B22:2/15  "OSR" %
% Rung: 23 %
SOR XIC B22:3/10 BST ADD 1.0 F8:47 F8:47 NXB MOV 0.0 F8:12 BND EOR
%   B22:3/10  "UNIT B ONGOING SERVICE FLOW CTR IS GREATER THAN 1 MILLION OSR" %
%   F8:47  "B SERVICE MILLIONS" %
%   F8:12  "B SERVICE THOUSANDS" %
% Rung: 24 %
SOR XIC B22:2/15 BST ADD 1.0 F8:38 F8:38 NXB MOV 0.0 F8:37 BND EOR
%   B22:2/15  "OSR" %
%   F8:38  B_REG_MIL %
%   F8:37  B_REG_THOU %
% Rung: 25 %
SOR GEQ F8:6 1000000 OSR B22:3/12 B22:3/13 EOR
%   F8:6  "B BATCH THOUSANDS" %
%   B22:3/12  "OSR FLOW MATH" %
%   B22:3/13  "OSR FLOW MATH2" %
% Rung: 26 %
SOR XIC B22:3/13 BST ADD 1.0 F8:49 F8:49 NXB MOV 0.0 F8:6 BND EOR
%   B22:3/13  "OSR FLOW MATH2" %
%   F8:49  "B BATCH MILLIONS" %
%   F8:6  "B BATCH THOUSANDS" %
% Rung: 27 %
SOR BST XIC B3:6/15 NXB GRT F8:47 999999 BND MOV 0.0 F8:47 EOR
%   B3:6/15  "RESET TOTALS DELAY FROM ALM SILENCE FOR 10 SECS" %
%   F8:47  "B SERVICE MILLIONS" %

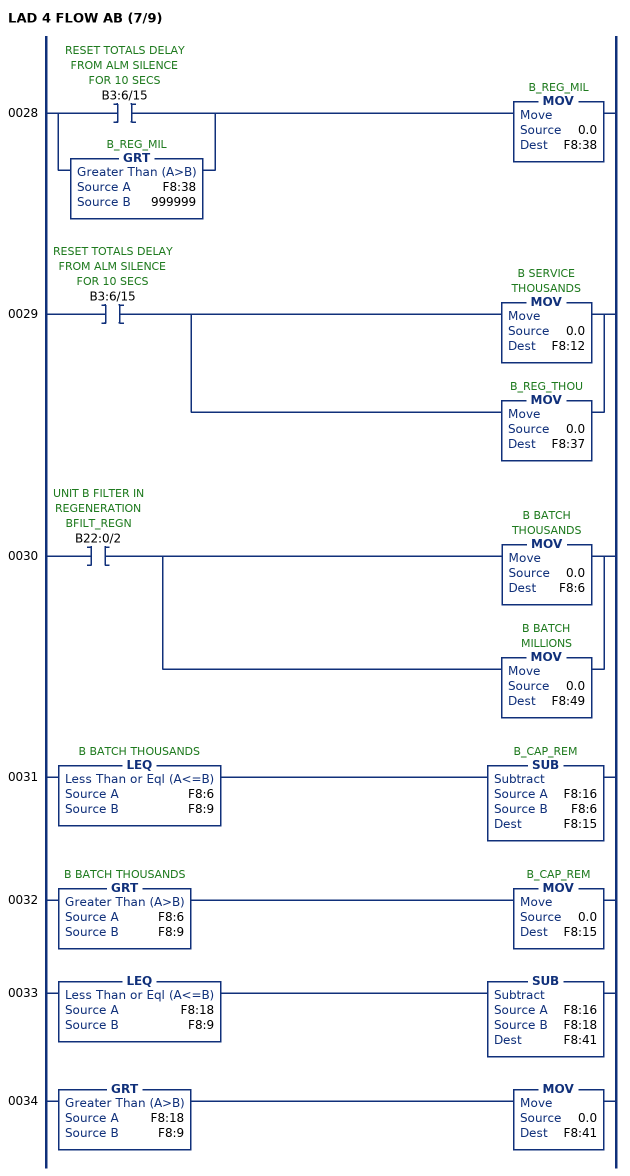
% Rung: 28 %
SOR BST XIC B3:6/15 NXB GRT F8:38 999999 BND MOV 0.0 F8:38 EOR
%   B3:6/15  "RESET TOTALS DELAY FROM ALM SILENCE FOR 10 SECS" %
%   F8:38  B_REG_MIL %
% Rung: 29 %
SOR XIC B3:6/15 BST MOV 0.0 F8:12 NXB MOV 0.0 F8:37 BND EOR
%   B3:6/15  "RESET TOTALS DELAY FROM ALM SILENCE FOR 10 SECS" %
%   F8:12  "B SERVICE THOUSANDS" %
%   F8:37  B_REG_THOU %
% Rung: 30 %
SOR XIC B22:0/2 BST MOV 0.0 F8:6 NXB MOV 0.0 F8:49 BND EOR
%   B22:0/2  BFILT_REGN  "UNIT B FILTER IN REGENERATION" %
%   F8:6  "B BATCH THOUSANDS" %
%   F8:49  "B BATCH MILLIONS" %
% Rung: 31 %
SOR LEQ F8:6 F8:9 SUB F8:16 F8:6 F8:15 EOR
%   F8:6  "B BATCH THOUSANDS" %
%   F8:9  "BATCH ENTRY FOR BATCH START" %
%   F8:16  T_GAL %
%   F8:15  B_CAP_REM %
% Rung: 32 %
SOR GRT F8:6 F8:9 MOV 0.0 F8:15 EOR
%   F8:6  "B BATCH THOUSANDS" %
%   F8:9  "BATCH ENTRY FOR BATCH START" %
%   F8:15  B_CAP_REM %
% Rung: 33 %
SOR LEQ F8:18 F8:9 SUB F8:16 F8:18 F8:41 EOR
%   F8:9  "BATCH ENTRY FOR BATCH START" %
%   F8:16  T_GAL %
% Rung: 34 %
SOR GRT F8:18 F8:9 MOV 0.0 F8:41 EOR
%   F8:9  "BATCH ENTRY FOR BATCH START" %

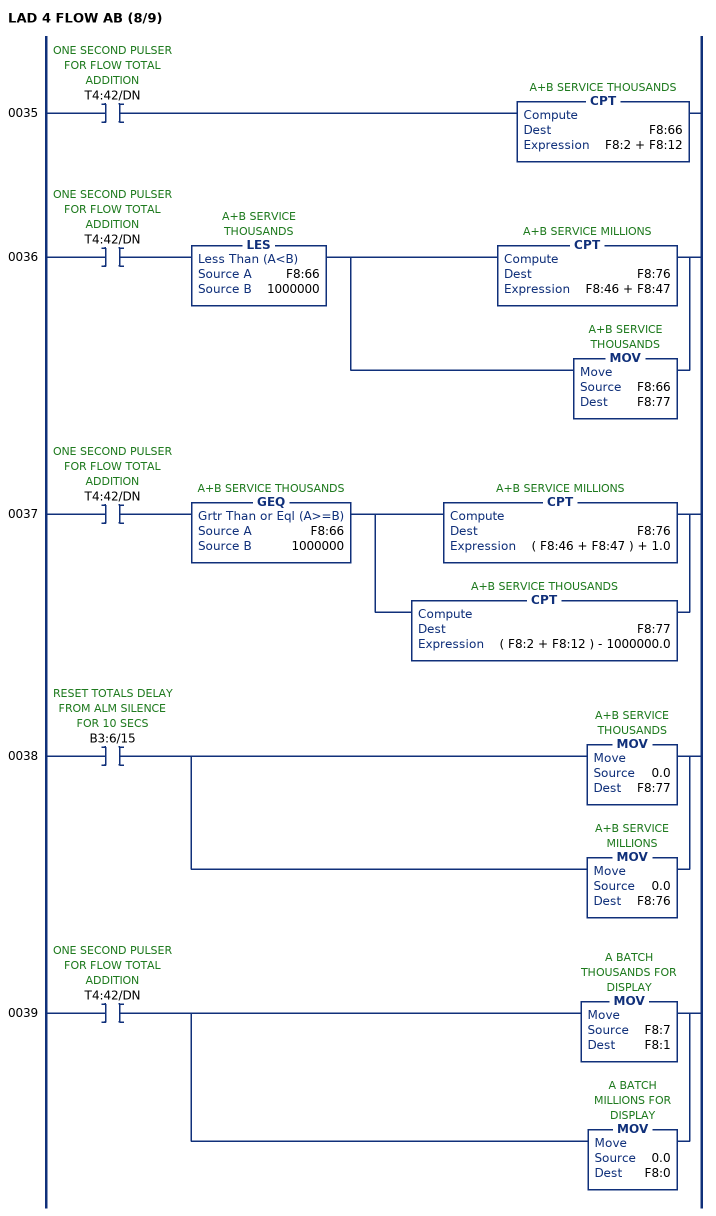
% Rung: 35 %
SOR XIC T4:42/DN CPT F8:66 " F8:2 + F8:12 " EOR
%   T4:42  "ONE SECOND PULSER FOR FLOW TOTAL ADDITION" %
%   F8:66  "A+B SERVICE THOUSANDS" %
%   F8:2  "A SERVICE THOUSANDS" %
%   F8:12  "B SERVICE THOUSANDS" %
% Rung: 36 %
SOR XIC T4:42/DN LES F8:66 1000000 BST CPT F8:76 " F8:46 + F8:47 " NXB MOV F8:66 F8:77 BND EOR
%   T4:42  "ONE SECOND PULSER FOR FLOW TOTAL ADDITION" %
%   F8:66  "A+B SERVICE THOUSANDS" %
%   F8:76  "A+B SERVICE MILLIONS" %
%   F8:46  "A SERVICE MILLIONS" %
%   F8:47  "B SERVICE MILLIONS" %
%   F8:77  "A+B SERVICE THOUSANDS" %
% Rung: 37 %
SOR XIC T4:42/DN GEQ F8:66 1000000 BST CPT F8:76 " ( F8:46 + F8:47 ) + 1.0 " NXB CPT F8:77 " ( F8:2 + F8:12 ) - 1000000.0 " BND EOR
%   T4:42  "ONE SECOND PULSER FOR FLOW TOTAL ADDITION" %
%   F8:66  "A+B SERVICE THOUSANDS" %
%   F8:76  "A+B SERVICE MILLIONS" %
%   F8:46  "A SERVICE MILLIONS" %
%   F8:47  "B SERVICE MILLIONS" %
%   F8:77  "A+B SERVICE THOUSANDS" %
%   F8:2  "A SERVICE THOUSANDS" %
%   F8:12  "B SERVICE THOUSANDS" %
% Rung: 38 %
SOR XIC B3:6/15 BST MOV 0.0 F8:77 NXB MOV 0.0 F8:76 BND EOR
%   B3:6/15  "RESET TOTALS DELAY FROM ALM SILENCE FOR 10 SECS" %
%   F8:77  "A+B SERVICE THOUSANDS" %
%   F8:76  "A+B SERVICE MILLIONS" %
% Rung: 39 %
SOR XIC T4:42/DN BST MOV F8:7 F8:1 NXB MOV 0.0 F8:0 BND EOR
%   T4:42  "ONE SECOND PULSER FOR FLOW TOTAL ADDITION" %
%   F8:7  "A BATCH THOUSANDS" %
%   F8:1  "A BATCH THOUSANDS FOR DISPLAY" %
%   F8:0  "A BATCH MILLIONS FOR DISPLAY" %

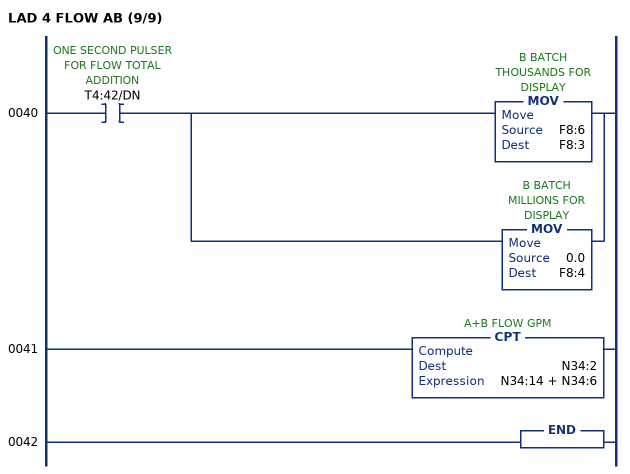
% Rung: 40 %
SOR XIC T4:42/DN BST MOV F8:6 F8:3 NXB MOV 0.0 F8:4 BND EOR
%   T4:42  "ONE SECOND PULSER FOR FLOW TOTAL ADDITION" %
%   F8:6  "B BATCH THOUSANDS" %
%   F8:3  "B BATCH THOUSANDS FOR DISPLAY" %
%   F8:4  "B BATCH MILLIONS FOR DISPLAY" %
% Rung: 41 %
SOR CPT N34:2 " N34:14 + N34:6 " EOR
%   N34:2  "A+B FLOW GPM" %
%   N34:14  AGPM  "FILTER A FLOW RATE" %
%   N34:6  BGPM  "UNIT B FLOW RATE" %
% Rung: 42 %
SOR END EOR

LADDER 5 "ALARMS"
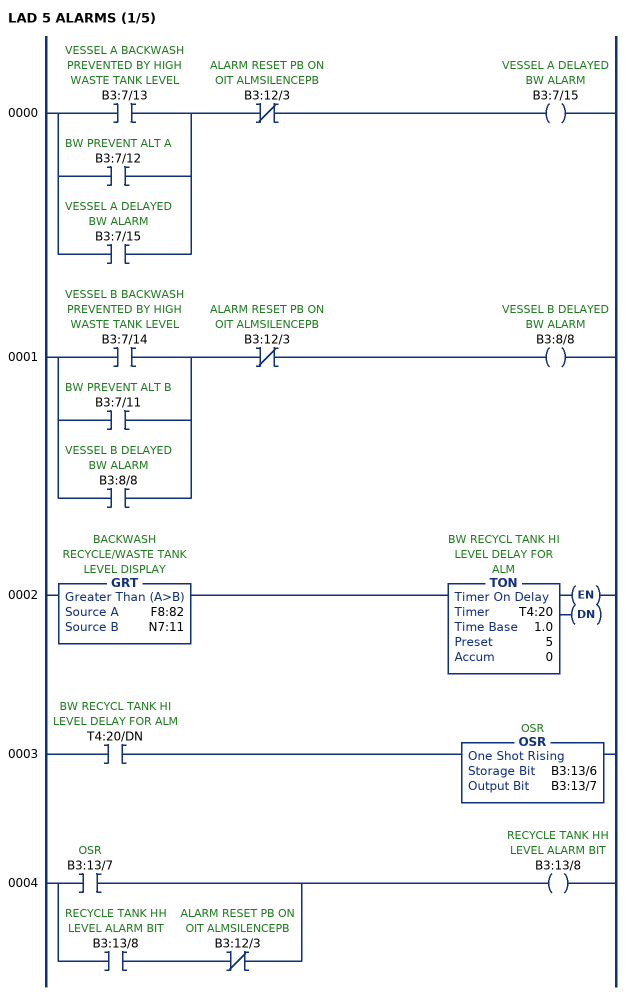
% Rung: 0 %
SOR BST XIC B3:7/13 NXB XIC B3:7/12 NXB XIC B3:7/15 BND XIO B3:12/3 OTE B3:7/15 EOR
%   B3:7/13  "VESSEL A BACKWASH PREVENTED BY HIGH WASTE TANK LEVEL" %
%   B3:7/12  "BW PREVENT ALT A" %
%   B3:7/15  "VESSEL A DELAYED BW ALARM" %
%   B3:12/3  ALMSILENCEPB  "ALARM RESET PB ON OIT" %
% Rung: 1 %
SOR BST XIC B3:7/14 NXB XIC B3:7/11 NXB XIC B3:8/8 BND XIO B3:12/3 OTE B3:8/8 EOR
%   B3:7/14  "VESSEL B BACKWASH PREVENTED BY HIGH WASTE TANK LEVEL" %
%   B3:7/11  "BW PREVENT ALT B" %
%   B3:8/8  "VESSEL B DELAYED BW ALARM" %
%   B3:12/3  ALMSILENCEPB  "ALARM RESET PB ON OIT" %
% Rung: 2 %
SOR GRT F8:82 N7:11 TON T4:20 1.0 5 0 EOR
%   F8:82  "BACKWASH RECYCLE/WASTE TANK LEVEL DISPLAY" %
%   N7:11  "BW RECYCLE TANK HIGH LEVEL ALM ENTRY" %
%   T4:20  "BW RECYCL TANK HI LEVEL DELAY FOR ALM" %
% Rung: 3 %
SOR XIC T4:20/DN OSR B3:13/6 B3:13/7 EOR
%   T4:20  "BW RECYCL TANK HI LEVEL DELAY FOR ALM" %
%   B3:13/6  "OSR" %
%   B3:13/7  "OSR" %
% Rung: 4 %
SOR BST XIC B3:13/7 NXB XIC B3:13/8 XIO B3:12/3 BND OTE B3:13/8 EOR
%   B3:13/7  "OSR" %
%   B3:13/8  "RECYCLE TANK HH LEVEL ALARM BIT" %
%   B3:12/3  ALMSILENCEPB  "ALARM RESET PB ON OIT" %

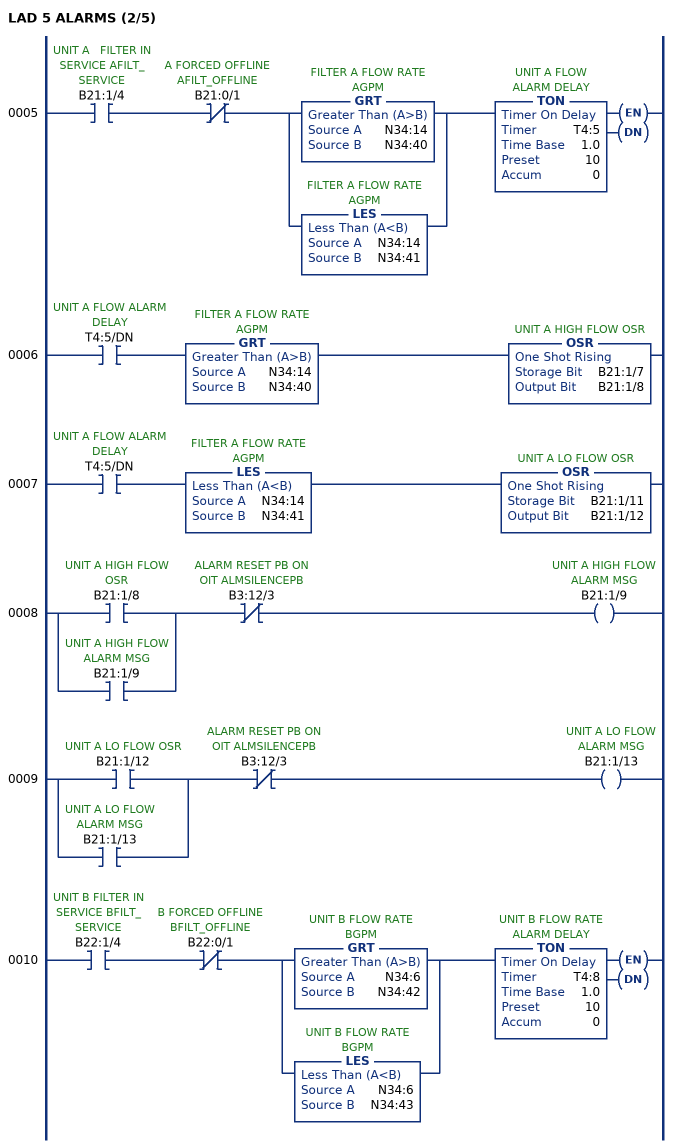
% Rung: 5 %
SOR XIC B21:1/4 XIO B21:0/1 BST GRT N34:14 N34:40 NXB LES N34:14 N34:41 BND TON T4:5 1.0 10 0 EOR
%   B21:1/4  AFILT_SERVICE  "UNIT A   FILTER IN SERVICE" %
%   B21:0/1  AFILT_OFFLINE  "A FORCED OFFLINE" %
%   N34:14  AGPM  "FILTER A FLOW RATE" %
%   N34:40  "UNIT A HIGH FLOW RATE SETPOINT FROM OIT" %
%   N34:41  "UNIT A LOW FLOW RATE SETPOINT FROM OIT" %
%   T4:5  "UNIT A FLOW ALARM DELAY" %
% Rung: 6 %
SOR XIC T4:5/DN GRT N34:14 N34:40 OSR B21:1/7 B21:1/8 EOR
%   T4:5  "UNIT A FLOW ALARM DELAY" %
%   N34:14  AGPM  "FILTER A FLOW RATE" %
%   N34:40  "UNIT A HIGH FLOW RATE SETPOINT FROM OIT" %
%   B21:1/7  "UNIT A HIGH FLOW OSR" %
%   B21:1/8  "UNIT A HIGH FLOW OSR" %
% Rung: 7 %
SOR XIC T4:5/DN LES N34:14 N34:41 OSR B21:1/11 B21:1/12 EOR
%   T4:5  "UNIT A FLOW ALARM DELAY" %
%   N34:14  AGPM  "FILTER A FLOW RATE" %
%   N34:41  "UNIT A LOW FLOW RATE SETPOINT FROM OIT" %
%   B21:1/11  "UNIT A LO FLOW OSR" %
%   B21:1/12  "UNIT A LO FLOW OSR" %
% Rung: 8 %
SOR BST XIC B21:1/8 NXB XIC B21:1/9 BND XIO B3:12/3 OTE B21:1/9 EOR
%   B21:1/8  "UNIT A HIGH FLOW OSR" %
%   B21:1/9  "UNIT A HIGH FLOW ALARM MSG" %
%   B3:12/3  ALMSILENCEPB  "ALARM RESET PB ON OIT" %
% Rung: 9 %
SOR BST XIC B21:1/12 NXB XIC B21:1/13 BND XIO B3:12/3 OTE B21:1/13 EOR
%   B21:1/12  "UNIT A LO FLOW OSR" %
%   B21:1/13  "UNIT A LO FLOW ALARM MSG" %
%   B3:12/3  ALMSILENCEPB  "ALARM RESET PB ON OIT" %
% Rung: 10 %
SOR XIC B22:1/4 XIO B22:0/1 BST GRT N34:6 N34:42 NXB LES N34:6 N34:43 BND TON T4:8 1.0 10 0 EOR
%   B22:1/4  BFILT_SERVICE  "UNIT B FILTER IN SERVICE" %
%   B22:0/1  BFILT_OFFLINE  "B FORCED OFFLINE" %
%   N34:6  BGPM  "UNIT B FLOW RATE" %
%   N34:42  "UNIT B HIGH FLOW RATE SETPOINT FROM OIT" %
%   N34:43  "UNIT B LOW FLOW ALARM SETPOINT FROM OIT" %
%   T4:8  "UNIT B FLOW RATE ALARM DELAY" %

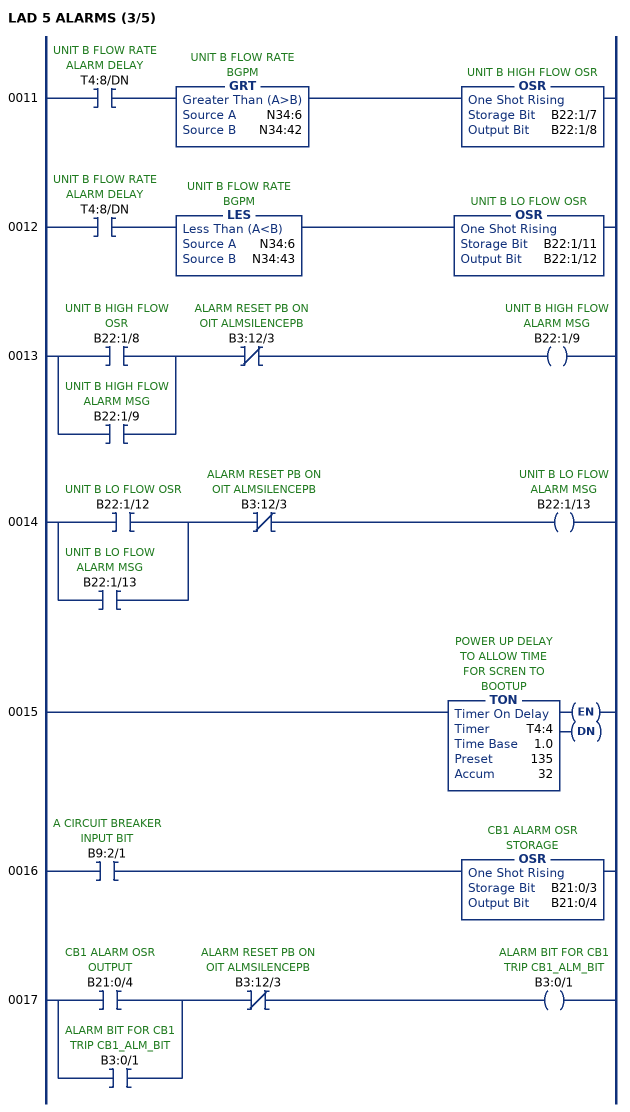
% Rung: 11 %
SOR XIC T4:8/DN GRT N34:6 N34:42 OSR B22:1/7 B22:1/8 EOR
%   T4:8  "UNIT B FLOW RATE ALARM DELAY" %
%   N34:6  BGPM  "UNIT B FLOW RATE" %
%   N34:42  "UNIT B HIGH FLOW RATE SETPOINT FROM OIT" %
%   B22:1/7  "UNIT B HIGH FLOW OSR" %
%   B22:1/8  "UNIT B HIGH FLOW OSR" %
% Rung: 12 %
SOR XIC T4:8/DN LES N34:6 N34:43 OSR B22:1/11 B22:1/12 EOR
%   T4:8  "UNIT B FLOW RATE ALARM DELAY" %
%   N34:6  BGPM  "UNIT B FLOW RATE" %
%   N34:43  "UNIT B LOW FLOW ALARM SETPOINT FROM OIT" %
%   B22:1/11  "UNIT B LO FLOW OSR" %
%   B22:1/12  "UNIT B LO FLOW OSR" %
% Rung: 13 %
SOR BST XIC B22:1/8 NXB XIC B22:1/9 BND XIO B3:12/3 OTE B22:1/9 EOR
%   B22:1/8  "UNIT B HIGH FLOW OSR" %
%   B22:1/9  "UNIT B HIGH FLOW ALARM MSG" %
%   B3:12/3  ALMSILENCEPB  "ALARM RESET PB ON OIT" %
% Rung: 14 %
SOR BST XIC B22:1/12 NXB XIC B22:1/13 BND XIO B3:12/3 OTE B22:1/13 EOR
%   B22:1/12  "UNIT B LO FLOW OSR" %
%   B22:1/13  "UNIT B LO FLOW ALARM MSG" %
%   B3:12/3  ALMSILENCEPB  "ALARM RESET PB ON OIT" %
% Rung: 15 %
SOR TON T4:4 1.0 135 32 EOR
%   T4:4  "POWER UP DELAY TO ALLOW TIME FOR SCREN TO BOOTUP" %
% Rung: 16 %
SOR XIC B9:2/1 OSR B21:0/3 B21:0/4 EOR
%   B9:2/1  "A CIRCUIT BREAKER INPUT BIT" %
%   B21:0/3  "CB1 ALARM OSR STORAGE" %
%   B21:0/4  "CB1 ALARM OSR OUTPUT" %
% Rung: 17 %
SOR BST XIC B21:0/4 NXB XIC B3:0/1 BND XIO B3:12/3 OTE B3:0/1 EOR
%   B21:0/4  "CB1 ALARM OSR OUTPUT" %
%   B3:0/1  CB1_ALM_BIT  "ALARM BIT FOR CB1 TRIP" %
%   B3:12/3  ALMSILENCEPB  "ALARM RESET PB ON OIT" %

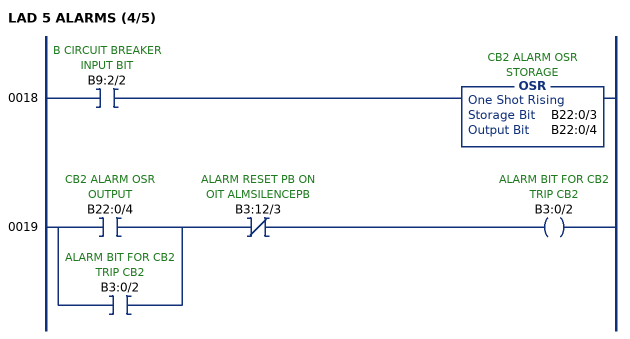
% Rung: 18 %
SOR XIC B9:2/2 OSR B22:0/3 B22:0/4 EOR
%   B9:2/2  "B CIRCUIT BREAKER INPUT BIT" %
%   B22:0/3  "CB2 ALARM OSR STORAGE" %
%   B22:0/4  "CB2 ALARM OSR OUTPUT" %
% Rung: 19 %
SOR BST XIC B22:0/4 NXB XIC B3:0/2 BND XIO B3:12/3 OTE B3:0/2 EOR
%   B22:0/4  "CB2 ALARM OSR OUTPUT" %
%   B3:0/2  CB2  "ALARM BIT FOR CB2 TRIP" %
%   B3:12/3  ALMSILENCEPB  "ALARM RESET PB ON OIT" %

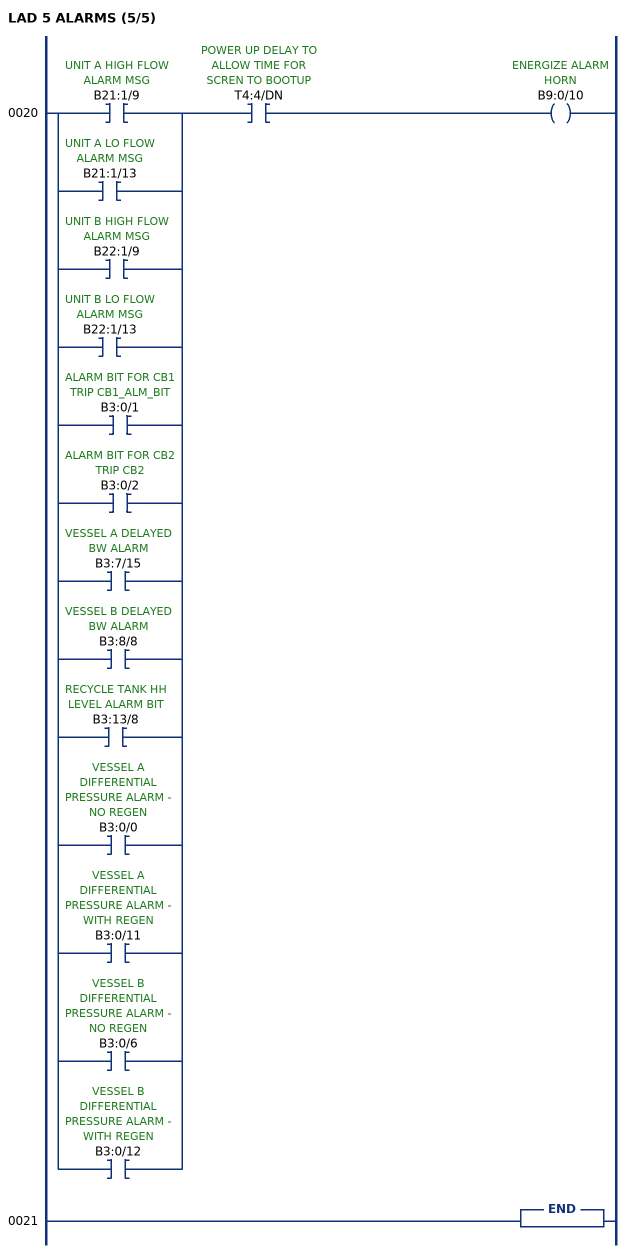
% Rung: 20 %
SOR BST XIC B21:1/9 NXB XIC B21:1/13 NXB XIC B22:1/9 NXB XIC B22:1/13 NXB XIC B3:0/1 NXB XIC B3:0/2 NXB XIC B3:7/15 NXB XIC B3:8/8 NXB XIC B3:13/8 NXB XIC B3:0/0 NXB XIC B3:0/11 NXB XIC B3:0/6 NXB XIC B3:0/12 BND XIC T4:4/DN OTE B9:0/10 EOR
%   B21:1/9  "UNIT A HIGH FLOW ALARM MSG" %
%   B21:1/13  "UNIT A LO FLOW ALARM MSG" %
%   B22:1/9  "UNIT B HIGH FLOW ALARM MSG" %
%   B22:1/13  "UNIT B LO FLOW ALARM MSG" %
%   B3:0/1  CB1_ALM_BIT  "ALARM BIT FOR CB1 TRIP" %
%   B3:0/2  CB2  "ALARM BIT FOR CB2 TRIP" %
%   B3:7/15  "VESSEL A DELAYED BW ALARM" %
%   B3:8/8  "VESSEL B DELAYED BW ALARM" %
%   B3:13/8  "RECYCLE TANK HH LEVEL ALARM BIT" %
%   B3:0/0  "VESSEL A DIFFERENTIAL PRESSURE ALARM - NO REGEN" %
%   B3:0/11  "VESSEL A DIFFERENTIAL PRESSURE ALARM - WITH REGEN" %
%   B3:0/6  "VESSEL B DIFFERENTIAL PRESSURE ALARM - NO REGEN" %
%   B3:0/12  "VESSEL B DIFFERENTIAL PRESSURE ALARM - WITH REGEN" %
%   T4:4  "POWER UP DELAY TO ALLOW TIME FOR SCREN TO BOOTUP" %
%   B9:0/10  "ENERGIZE ALARM HORN" %
% Rung: 21 %
SOR END EOR

LADDER 6 "TIME TRIG"    % TIME INTERVAL REGN INITIATION %
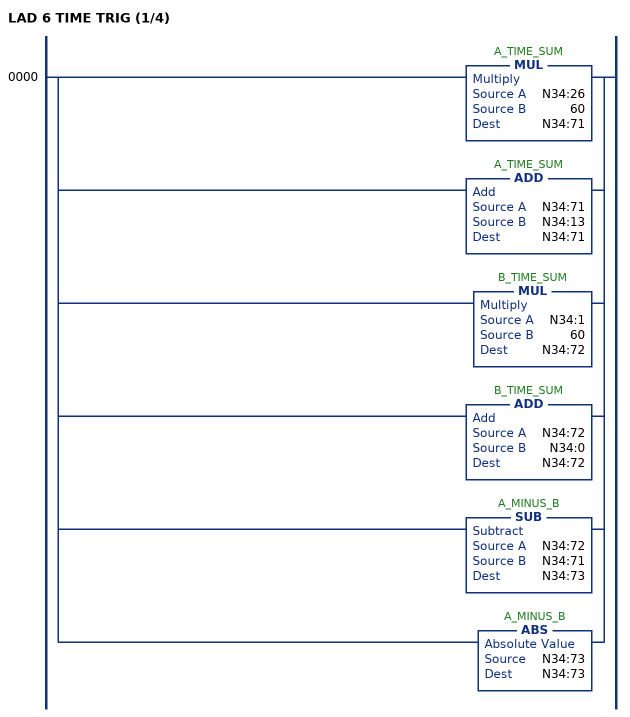
% Rung: 0 %
SOR BST MUL N34:26 60 N34:71 NXB ADD N34:71 N34:13 N34:71 NXB MUL N34:1 60 N34:72 NXB ADD N34:72 N34:0 N34:72 NXB SUB N34:72 N34:71 N34:73 NXB ABS N34:73 N34:73 BND EOR
%   N34:26  "FILTER A HOUR OF DAY TO START SELECT EITHER DUE TO BATCH OR ELAPSED TIME OR DP" %
%   N34:71  A_TIME_SUM %
%   N34:13  "FILTER A MIN OF DAY TO START SELECT EITHER DUE TO BATCH OR ELAPSED TIME" %
%   N34:1  "FILTER B HOUR OF DAY TO START SELECT EITHER DUE TO BATCH OR ELAPSED TIME OR DP" %
%   N34:72  B_TIME_SUM %
%   N34:0  "FILTER B MIN OF DAY TO START SELECT EITHER DUE TO BATCH OR ELAPSED TIME" %
%   N34:73  A_MINUS_B %

